// TIA Portal project "COENEXION S7-1200" (V11)

(* hardware
DEVICE "Estación SIMATIC 1200_1"  S71200.Device
   slot 0: "Rack S7-1200"  Rack  V1.0
   slot 1: "PLC_1"  CPU 1214C AC/DC/Rly  6ES7 214-1BE30-0XB0  V2.2
*)

// ===== PLC "PLC_1"  CPU 1214C AC/DC/Rly =====

ORGANIZATION_BLOCK "Main"   // OB1, LAD, ProgramCycle
TITLE = "Main Program Sweep (Cycle)"
{ S7_Optimized_Access := 'FALSE' }
VERSION : 0.1
BEGIN
END_ORGANIZATION_BLOCK